Universal Robots PolyScope program: rtde_2.urp

Program rtde_2 (createdIn=3.4.0.265 lastSavedIn=3.4.0.265 directory=/home/ur/ursim-current/programs/RTDE installation=rtde_ext robotSerialNumber=2014309999)
Calibrated DH parameters: a=[0, -0.612, -0.5723, 0, 0, 0]; d=[0.1273, 0, 0, 0.163941, 0.1157, 0.0922]; alpha=[1.570796, 0, 0, 1.570796, -1.570796, 0]; deltaTheta=[0, 0, 0, 0, 0, 0]
BeforeStart
  Script: write_output_integer_register(0, 0)
  MoveJ speed 60 deg/s, acceleration 80 deg/s^2 (useActiveTCP=false)
    Waypoint Waypoint_1: TCP in base x=-365.427 y=-608.045 z=138.208 mm, rx=-0.0328 ry=-0.0109 rz=-0.7431 rad; joints [45.22, -98.39, 96.77, 0.13, 87.82, -88.71] deg; flange x=-288.197 y=-528.14 z=635.664 mm, rx=1.7084 ry=0.7281 rz=-1.7369 rad
  Popup Message (haltProgram=false message=Start Script on PC now)
  SuppressedNode
    Script: set_tcp(p[0.5,-0.013529999999999999,0.09813,-1.2092,-1.2092,1.2092])
Robot Program (runOnlyOnce=true motionType=MoveJ speed=1.047198 acceleration=1.396263 useActiveTCP=false)
  Script file /home/ur/ursim-current/programs/RTDE/int
    | global setp=p[0,0,0,0,0,0]
    | global setp2=p[0,0,0,0,0,0]
    | global setp3=p[0,0,0,0,0,0]
    | global setp4=p[0,0,0,0,0,0]
    | global setp5=p[0,0,0,0,0,0]
    | global setp6=p[0,0,0,0,0,0]
    | global setp7=p[0,0,0,0,0,0]
    | global setp8=p[0,0,0,0,0,0]
    | global setp9=p[0,0,0,0,0,0]
    | global setp10=p[0,0,0,0,0,0]
    | global moveTo=p[0,0,0,0,0,0]
    | global speed=0.03
    | global zone=0.001
    | global tcp=p[0,0,0,0,0,0]
    | global weight = 0
    | global cog = [0,0,0]
    | global robotloc=0
    | global bufferFillLoc=0
    | listPoints=[setp,setp2,setp3,setp4,setp5,setp6,setp7,setp8,setp9,setp10]
    | listSpeeds=[0.03,0.03,0.03,0.03,0.03,0.03,0.03,0.03,0.03,0.03]
    | listZones=[0.001,0.001,0.001,0.001,0.001,0.001,0.001,0.001,0.001,0.001]
    | bufferStatus=[0,0,0,0,0,0,0,0,0,0]
    | rtde_set_watchdog("input_int_register_0", 1, "PAUSE")
    | write_output_integer_register(0, 0)
  Script file /home/ur/ursim-current/programs/RTDE/tcpsetup.script
    | keep_running = True
    | global loopcheck = 0
    | global loopcheck2 = 0
    | while keep_running:
    |   write_output_integer_register(0, 2)
    |   sync()
    |   sleep(2)
    |   global tmpTCP=p[0,0,0,0,0,0]
    |   tmpTCP[0] = read_input_float_register(7)
    |   tmpTCP[1] = read_input_float_register(8)
    |   tmpTCP[2] = read_input_float_register(9)
    |   tmpTCP[3] = read_input_float_register(10)
    |   tmpTCP[4] = read_input_float_register(11)
    |   tmpTCP[5] = read_input_float_register(12)
    |   loopcheck = loopcheck + 1
    |   if (tmpTCP != p[0,0,0,0,0,0]):
    |     loopcheck2 = loopcheck2 + 1
    |     tcp=tmpTCP
    |     global tmpWeight = 0
    |     tmpWeight = read_input_float_register(14)
    |     weight = tmpWeight
    |     global tmpCOG = [0,0,0]
    |     tmpCOG[0] = read_input_float_register(15)
    |     tmpCOG[1] = read_input_float_register(16)
    |     tmpCOG[2] = read_input_float_register(17)
    |     cog = tmpCOG
    |     keep_running = False
    |   end
    |   write_output_integer_register(0, 0)
    |   sync()
    | end
  Script file /home/ur/ursim-current/programs/RTDE/Thread_1
    |  thread Thread_1():
    |  while (True):
    |      sync()
    |      if (bufferStatus[bufferFillLoc]==0):
    |       write_output_integer_register(0, 1)
    |       sync()
    |       global tmp=p[0,0,0,0,0,0]
    |       tmp[0] = read_input_float_register(0)
    |       tmp[1] = read_input_float_register(1)
    |       tmp[2] = read_input_float_register(2)
    |       tmp[3] = read_input_float_register(3)
    |       tmp[4] = read_input_float_register(4)
    |       tmp[5] = read_input_float_register(5)
    |       listPoints[bufferFillLoc]=tmp
    |       speed = read_input_float_register(18)
    |       zone = read_input_float_register(19)
    |       bufferStatus[bufferFillLoc]=1
    |       bufferFillLoc=bufferFillLoc+1
    |       if (bufferFillLoc>9):
    |         bufferFillLoc=0
    |       end
    |       write_output_integer_register(0, 0)
    |       sync()
    |     end
    |   end
    | end
  Script: threadId_Thread_1 = run Thread_1()
  SuppressedNode
    Script: set_tcp(p[0.5,-0.013529999999999999,0.09813,-1.2092,-1.2092,1.2092])
  Script: set_tcp(tcp)
  Script: set_payload(weight, cog)
  Loop Forever
    Script file /home/ur/ursim-current/programs/RTDE/mainloop
      | if (bufferStatus[robotloc]==1):
      |       sync()
      |       global moveTo=listPoints[robotloc]
      |       movel(pose_trans(p[0.0,0.0,0.0,0.0,0.0,0.0], moveTo), a=1.2, v=0.03, r=0.001)
      |       bufferStatus[robotloc]=0
      |       robotloc=robotloc+1
      |       if (robotloc>9):
      |         robotloc=0
      |       end
      | else:
      |       sync()
      | end
      | sync()
    Script file /home/ur/ursim-current/programs/RTDE/varview.script
      | setp=listPoints[0]
      | setp2=listPoints[1]
      | setp3=listPoints[2]
      | setp4=listPoints[3]
      | setp5=listPoints[4]
      | setp6=listPoints[5]
      | setp7=listPoints[6]
      | setp8=listPoints[7]
      | setp9=listPoints[8]
      | setp10=listPoints[9]
  Script: write_output_integer_register(0, 3)
